    #fbManualMode(Enable := (#State = STATE_MANUAL), SelectedAxis := "DB_Manual".SelectedAxis,
                  Jog_Plus := "DB_Manual".Jog_Plus, Jog_Minus := "DB_Manual".Jog_Minus,
                  JogSpeed := "DB_Manual".JogSpeed,
                  MoveAbsolute := "DB_Manual".Btn_MoveAbsolute, TargetPosition := "DB_Manual".MoveToPosition,
                  HomeAxis := "DB_Manual".Btn_HomeAxis, HomeAll := "DB_Manual".Btn_HomeAll,
                  HomingMode := "DB_Manual".HomingMode, HomePosition := 0.0,
                  GoSafe := "DB_Manual".Btn_GoSafe, GoZero := "DB_Manual".Btn_GoZero,
                  SafeToJog := #fbSafetyMonitor.SafeToJog, Reset := #fbInputs.Cmd_Reset,
                  PNP_X_Min := #HW_PNP_X_Min, PNP_Z_Min := #HW_PNP_Z_Min,
                  ToolStepCW := "DB_Manual".Btn_ToolStepCW, ToolStepCCW := "DB_Manual".Btn_ToolStepCCW,
                  ToolStepAngle := "DB_Manual".ToolStepAngle, ToolStepSpeed := "DB_Manual".ToolStepSpeed,
                  Axis_X := #Axis_X, Axis_Z := #Axis_Z, Axis_Tool := #Axis_Tool, Axis_Spindle := #Axis_Spindle);

    // Update manual mode status
    "DB_Manual".JogBusy := #fbManualMode.Busy;
    "DB_Manual".ManualBusy := #fbManualMode.Busy;       // Alias
    "DB_Manual".JogError := #fbManualMode.Error;
    "DB_Manual".ManualError := #fbManualMode.Error;     // Alias
    "DB_Manual".JogErrorID := #fbManualMode.ErrorID;
    "DB_Manual".ManualErrorID := #fbManualMode.ErrorID; // Alias
    "DB_Manual".SelectedAxisPos := SEL(G := "DB_Manual".SelectedAxis = 0,
                                        IN0 := #Axis_Z.ActualPosition, IN1 := #Axis_X.ActualPosition);
    "DB_Manual".SelectedAxisName := SEL(G := "DB_Manual".SelectedAxis = 0, IN0 := 'Z', IN1 := 'X');
    "DB_Manual".ToolPosition := #Axis_Tool.ActualPosition;
    "DB_Manual".ActiveAxis := #fbManualMode.ActiveAxis;

    // Forward manual mode errors to alarm manager (once, on rising edge)
    IF #fbManualMode.Error AND NOT #prevManualError THEN
        #newErrorFlag := TRUE;
        #newErrorCode := #fbManualMode.ErrorID;
        // DB_HMI.ErrorDetail is written directly inside FB_ManualMode at each error point.
        // Write ErrorText here as a fallback for any code not yet handled with direct detail.
        "DB_HMI".ErrorText := 'Manual mode error - check ErrorDetail and ErrorID';
    END_IF;
    #prevManualError := #fbManualMode.Error;

    // =========================================================================
    // SPINDLE CONTROL
    // Manual mode spindle control via DB_Manual buttons
    // Recipe handler spindle control via bSpindleStart/bSpindleStop flags
    // =========================================================================
    #fbSpindleControl(
        Start := "DB_Manual".Btn_SpindleStart OR #bSpindleStart,
        Stop := "DB_Manual".Btn_SpindleStop OR #bSpindleStop OR #fbInputs.Cmd_Stop,
        SetSpeed := SEL(G := (#State = STATE_MANUAL),
                        IN0 := "DB_Spindle".Cmd_SetSpeed,
                        IN1 := "DB_Manual".Manual_SpindleSpeed),
        Direction := SEL(G := (#State = STATE_MANUAL),
                         IN0 := "DB_Spindle".Cmd_Direction,
                         IN1 := "DB_Manual".Manual_SpindleDir),
        SpeedOverride := "DB_Spindle".SpeedOverride,
        Reset := #fbInputs.Cmd_Reset,
        AckError := #ackEdge OR "DB_Manual".Btn_SpindleAckError,  // Main Ack or spindle-specific Ack (no full Reset needed)
        Axis_Spindle := #Axis_Spindle
    );

    // Diagnostic output
    "DB_Diagnostic".Process_State        := #State;
    "DB_Diagnostic".Process_SafeToRun    := #SafeToRun;
    "DB_Diagnostic".Process_DrivesEnable := #bDrivesEnable;
    "DB_Diagnostic".Recipe_CurrentProgram := #activeProgram;
    "DB_Diagnostic".Recipe_TotalLines    := #activeLineCount;
    "DB_Diagnostic".Axis_X_Pos           := #Axis_X.ActualPosition;
    "DB_Diagnostic".Axis_Z_Pos           := #Axis_Z.ActualPosition;
    "DB_Diagnostic".Axis_X_Enabled       := #fbPowerX.Status;
    "DB_Diagnostic".Axis_Z_Enabled       := #fbPowerZ.Status;
    "DB_Diagnostic".Axis_X_Homed         := #Axis_X.StatusBits.HomingDone;
    "DB_Diagnostic".Axis_Z_Homed         := #Axis_Z.StatusBits.HomingDone;

    // =========================================================================
    // CONTACTOR CONTROL -- called as the last step of FB_Process.
    // FC_ContactorControl reads DB_HMI.Btn_Contactor_* and Bypass_EStop/HasError.
    // In auto mode STATE_STARTING already sets these flags TRUE; they are reflected to I/O here.
    // Called here rather than from OB1 to ensure contactor logic runs in sync with the process.
    // =========================================================================
    "FC_ContactorControl"();
END_FUNCTION_BLOCK
